{attribute 'linkalways'} 
{attribute 'no_explicit_call' := 'This FB is a CLASS and must be accessed using methods or properties'}
{attribute 'enable_dynamic_creation'}
FUNCTION_BLOCK Node_F_VN_DrawLine EXTENDS VisionNode
VAR
    nX1 : _UDINT(0);
    nY1 : _UDINT(0);
    nX2 : _UDINT(0);
    nY2 : _UDINT(0);
    ipDestImage : _ITcVnImage;
    aColor : _TcVnVector4_LREAL;
    nThickness : _DINT(1);
    hrPrev : _HRESULT(S_OK);
	hresult : _HRESULT(S_OK);
END_VAR

METHOD PUBLIC  Clone : I_Node
VAR
	pNode : POINTER TO Node_F_VN_DrawLine;
END_VAR
pNode := __NEW(Node_F_VN_DrawLine);
Clone := pNode^;
END_METHOD

METHOD FB_init : BOOL
VAR_INPUT
	bInitRetains : BOOL; // if TRUE, the retain variables are initialized (warm start / cold start)
	bInCopyCode : BOOL;  // if TRUE, the instance afterwards gets moved into the copy code (online change)
END_VAR
AddParameter('nX1', nX1);
AddParameter('nY1', nY1);
AddParameter('nX2', nX2);
AddParameter('nY2', nY2);
AddInput('ipDestImage', ipDestImage);
AddInput('aColor', aColor);
AddParameter('nThickness', nThickness);
AddInput('hrPrev', hrPrev);
AddOutput('ipDestImage', ipDestImage);
AddOutput('hresult',hresult);
END_METHOD

METHOD PROTECTED OnExecute
hresult.Value := F_VN_DrawLine(
    nX1 := nX1.Value,
    nY1 := nY1.Value,
    nX2 := nX2.Value,
	nY2 := nY2.Value,
	ipDestImage := ipDestImage.Value,
    aColor := aColor.Value,
    nThickness := nThickness.Value,
	hrPrev:= hrPrev.Value);
END_METHOD

METHOD PUBLIC PreExecutionCheck
VAR_INPUT
	Check : I_PreExecutionChecks;
END_VAR
Check.IsTrue(ipDestImage.IsValid, 'ipDestImage must contain an image');
Check.IsTrue(nThickness.Value >= 1, 'nThickness must be greater than or equal to 1');
END_METHOD

END_FUNCTION_BLOCK

(* stored: Version 1.1.0.1, ProductVersion 3.1.4024.15
   POU Node_F_VN_DrawLine: Id {dc653c7a-2933-0576-2626-1faa874c03b0}, SpecialFunc None
   Folder Constructor: Id {a5913828-a77a-0588-0b42-01dc512a4cf4}
   Method Clone: Id {d264fbd2-1fc9-0a2c-339a-46b0e119c9a0}
   Method FB_init: Id {ce37e974-3225-0748-34f6-48f40a96ea5a}
   Method OnExecute: Id {40947ae6-2476-0427-1850-8226b5b7e1bd}
   Method PreExecutionCheck: Id {8aab7573-0bc6-0ee8-1b5e-66d20084a33b} *)
